FUNCTION_BLOCK BoolValueChanged_6 (* Basic Function Block Type *)
  (* Standard: 61499-2 *)
  (* Version 0.0, 6/25/2026, Schneider Electric, Template *)
  PACKAGE SE.Nereda;
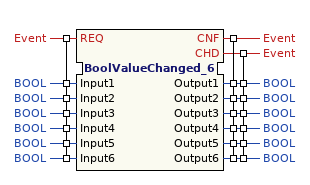
  EVENT_INPUT
    REQ WITH Input1, Input2, Input3, Input4, Input5, Input6; (* Normal Execution Request *)
  END_EVENT
  EVENT_OUTPUT
    CNF WITH Output1, Output2, Output3, Output4, Output5, Output6; (* Execution Confirmation *)
    CHD WITH Output2, Output3, Output4, Output5, Output6, Output1;
  END_EVENT
  VAR_INPUT
    Input1 : BOOL; (* Input event qualifier *)
    Input2 : BOOL;
    Input3 : BOOL;
    Input4 : BOOL;
    Input5 : BOOL;
    Input6 : BOOL;
  END_VAR
  VAR_OUTPUT
    Output1 : BOOL; (* Output event qualifier *)
    Output2 : BOOL;
    Output3 : BOOL;
    Output4 : BOOL;
    Output5 : BOOL;
    Output6 : BOOL;
  END_VAR
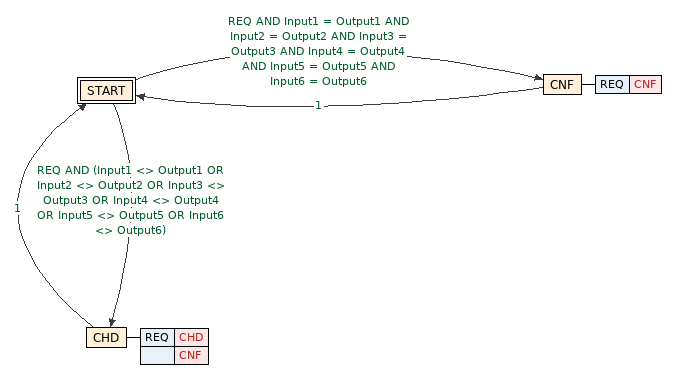
  EC_STATES
    START; (* Initial State *)
    CNF : REQ -> CNF;
    CHD : REQ -> CHD, -> CNF;
  END_STATES
  EC_TRANSITIONS
    CHD TO START := 1;
    CNF TO START := 1;
    START TO CHD := REQ AND (Input1 <> Output1 OR Input2 <> Output2 OR Input3 <> Output3 OR Input4 <> Output4 OR Input5 <> Output5 OR Input6 <> Output6);
    START TO CNF := REQ AND Input1 = Output1 AND Input2 = Output2 AND Input3 = Output3 AND Input4 = Output4 AND Input5 = Output5 AND Input6 = Output6;
  END_TRANSITIONS
  ALGORITHM REQ IN ST: (* Normally executed algorithm *)
;
Output1 := Input1;
Output2 := Input2;
Output3 := Input3;
Output4 := Input4;
Output5 := Input5;
Output6 := Input6;
  END_ALGORITHM
END_FUNCTION_BLOCK
